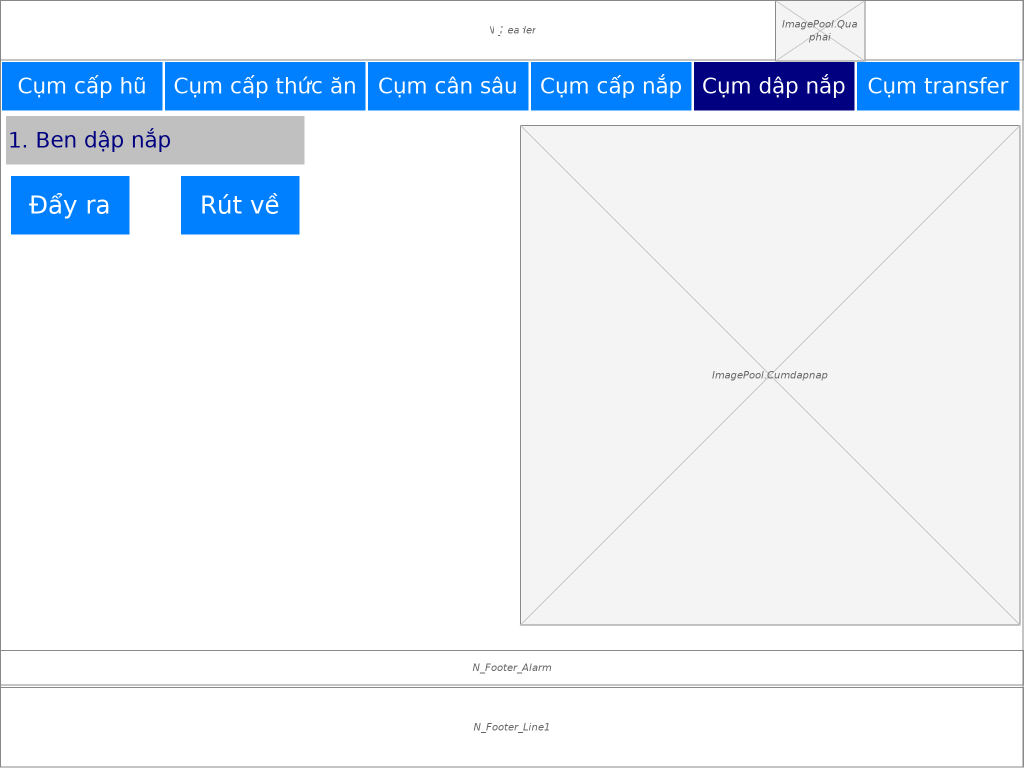
VISUALIZATION N_LidPressing1  // 1024x768
    Rectangle (180,175 120x60), "Rút về", colour toggle: PR_Line01.bCylinder_CloseLid_Retract
        OnMouseDown: execute { PR_Line01.bCylinder_CloseLid_Retract := TRUE; PR_Line01.bCylinder_CloseLid_Extend := FALSE; }
    Frame (0,687 1024x80)
        shows N_Footer_Line1()
    Frame (0,0 1024x60)
        shows N_Header()
    Textfield (353,5 400x50), "MÀN HÌNH CHẠY TAY LINE 1"
    Rectangle (5,115 300x50), "1. Ben dập nắp"
    Rectangle (10,175 120x60), "Đẩy ra", colour toggle: PR_Line01.bCylinder_CloseLid_Extend
        OnMouseDown: execute { PR_Line01.bCylinder_CloseLid_Extend := TRUE; PR_Line01.bCylinder_CloseLid_Retract := FALSE; }
    Rectangle (1,61 162x50), "Cụm cấp hũ"
        OnMouseClick: change screen: N_JarSupply1
    Rectangle (164,61 202x50), "Cụm cấp thức ăn"
        OnMouseClick: change screen: N_FoodSupply1
    Rectangle (367,61 162x50), "Cụm cân sâu"
        OnMouseClick: change screen: N_WormWeight1
    Rectangle (530,61 162x50), "Cụm cấp nắp"
        OnMouseClick: change screen: N_LidSupply1
    Rectangle (693,61 162x50), "Cụm dập nắp"
        OnMouseClick: change screen: N_LidPressing1
    Rectangle (856,61 164x50), "Cụm transfer"
        OnMouseClick: change screen: N_Tranfer1
    Image (775,0 90x61), input disabled if: bResetAuto2, image: ImagePool.Qua phai
        OnMouseClick: change screen: N_LidPressing2
        OnMouseClick: execute { MAIN_LINE2.bModeManual := TRUE; MAIN_LINE2.bModeAuto := FALSE; }
    Image (520,125 500x500), image: ImagePool.Cumdapnap
    Frame (0,650 1024x35)
        shows N_Footer_Alarm()
END_VISUALIZATION

(* stored: Version 1.1.0.1, ProductVersion 3.1.4024.12
   Visu N_LidPressing1: Id {727139d6-cfa1-40ba-834b-c9e8fe6ad3b6} *)
